TYPE ST_Event :
STRUCT
    eEventType: E_EventType;
	eEventSeverity: TcEventSeverity;
	nEventIdentity : UDINT;
	sEventText: STRING(255);
	dtTimeStamp: DATE_AND_TIME;
	
END_STRUCT
END_TYPE

(* stored: Version 1.1.0.1, ProductVersion 3.1.4024.12
   DUT ST_Event: Id {b1e3ceb9-a389-4007-a41f-58ed9396e74e} *)
